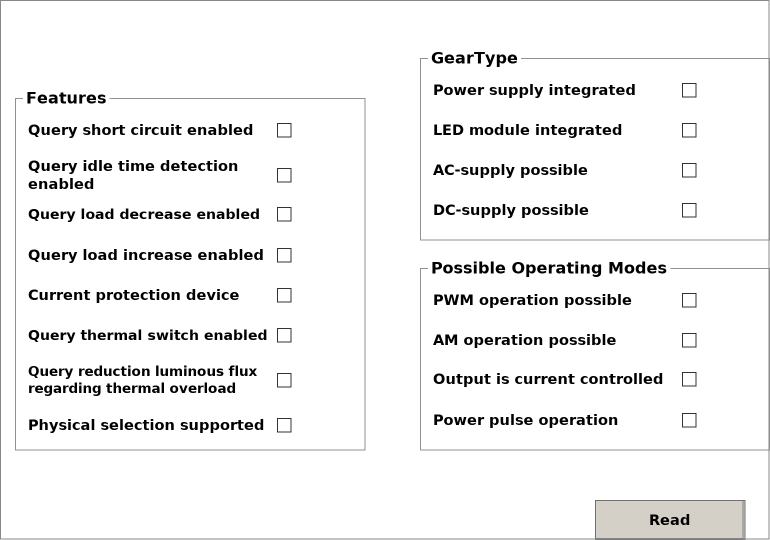
VISUALIZATION Visu_Part207Parameters  // 770x540
    Button (595,500 150x40), "Read"
        OnMouseClick: execute { DALI_Commissioning.fbPart207LED.bReadParameter:=TRUE; }
    GroupBox (420,50 350x190), "GearType"
        Textfield (10,25 220x30), "Power supply integrated"
        Checkbox (260,25 30x30), variable: DALI_Commissioning.fbPart207LED.bLEDPowerSupply, input disabled if: True
        Textfield (10,65 220x30), "LED module integrated"
        Textfield (10,145 220x30), "DC-supply possible"
        Textfield (10,105 220x30), "AC-supply possible"
        Checkbox (260,65 30x30), variable: DALI_Commissioning.fbPart207LED.bLEDModule, input disabled if: True
        Checkbox (260,145 30x30), variable: DALI_Commissioning.fbPart207LED.bDCSupply, input disabled if: True
        Checkbox (260,105 30x30), variable: DALI_Commissioning.fbPart207LED.bACSupply, input disabled if: True
    GroupBox (15,90 350x360), "Features"
        Textfield (10,25 240x30), "Query short circuit enabled"
        Checkbox (260,25 30x30), variable: DALI_Commissioning.fbPart207LED.bQueryShortCircuitEnabled, input disabled if: True
        Textfield (10,65 240x40), "Query idle time detection enabled"
        Textfield (10,150 240x30), "Query load increase enabled"
        Textfield (10,109 240x30), "Query load decrease enabled"
        Checkbox (260,70 30x30), variable: DALI_Commissioning.fbPart207LED.bQueryIdleTimeDetectionEnabled, input disabled if: True
        Checkbox (260,150 30x30), variable: DALI_Commissioning.fbPart207LED.bQueryLoadIncreaseEnabled, input disabled if: True
        Checkbox (260,109 30x30), variable: DALI_Commissioning.fbPart207LED.bQueryLoadDecreaseEnabled, input disabled if: True
        Textfield (10,190 240x30), "Current protection device"
        Checkbox (260,190 30x30), variable: DALI_Commissioning.fbPart207LED.bQueryCurrentProtectionDevicePresent, input disabled if: True
        Checkbox (260,230 30x30), variable: DALI_Commissioning.fbPart207LED.bQueryThermalSwitchEnabled, input disabled if: True
        Checkbox (260,275 30x30), variable: DALI_Commissioning.fbPart207LED.bQueryReductionOfLuminouFluxRegardingThermalOverloadEnabled, input disabled if: True
        Checkbox (260,320 30x30), variable: DALI_Commissioning.fbPart207LED.bPhysicalSelectionSupported, input disabled if: True
        Textfield (10,230 240x30), "Query thermal switch enabled"
        Textfield (10,270 240x40), "Query reduction luminous flux regarding thermal overload"
        Textfield (10,320 240x30), "Physical selection supported"
    GroupBox (420,260 350x190), "Possible Operating Modes", invisible if: DALI_Commissioning.fbPart207LED.bInvisible
        Checkbox (260,25 30x30), variable: DALI_Commissioning.fbPart207LED.bPWMOperation, input disabled if: True
        Textfield (10,65 240x30), "AM operation possible"
        Textfield (10,145 240x30), "Power pulse operation"
        Textfield (10,104 240x30), "Output is current controlled"
        Checkbox (260,65 30x30), variable: DALI_Commissioning.fbPart207LED.bAMOperation, input disabled if: True
        Checkbox (260,145 30x30), variable: DALI_Commissioning.fbPart207LED.bPowerPulseOperation, input disabled if: True
        Checkbox (260,104 30x30), variable: DALI_Commissioning.fbPart207LED.bOutputCurrentControlled, input disabled if: True
        Textfield (10,25 240x30), "PWM operation possible"
END_VISUALIZATION

(* stored: Version 1.1.0.1, ProductVersion 3.1.4024.12
   Visu Visu_Part207Parameters: Id {4da47d3e-8855-4f6c-a557-60855b37564a} *)
